Yaskawa INFORM job: BATMAN_4SPOINY.JBI

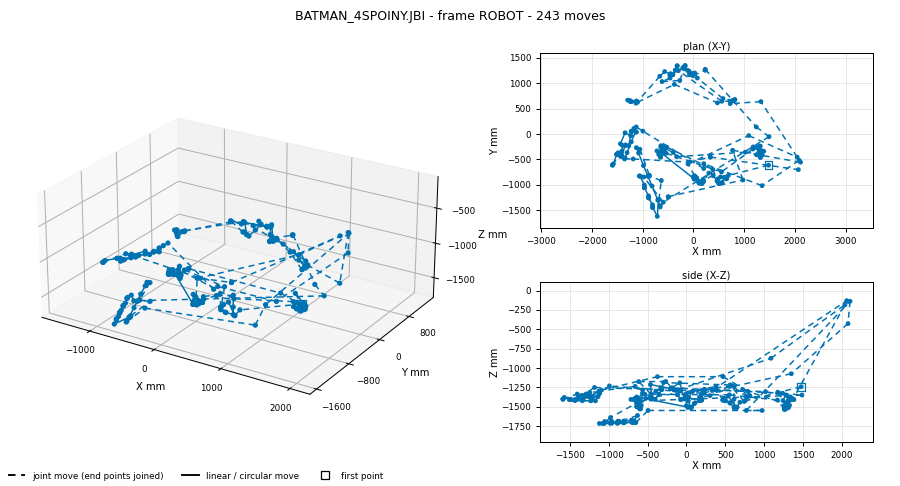
[picture p0: tool path of BATMAN_4SPOINY.JBI in frame ROBOT, 243 of 243 moves have a stored position in this frame; points joined in program order, loops and branches not executed]
/JOB
//NAME BATMAN_4SPOINY
///FOLDERNAME KRIS-SCIANA
//POS
///NPOS 293,293,243,19,0,0
///TOOL 0
///POSTYPE ROBOT
///RECTAN
///RCONF 0,0,0,0,0,0,0,0,0,0,0,0,0,0,0,0,0,0,0,0,0,0,0,0
C00000=1479.209,-614.254,-1239.827,11.6326,33.9671,-178.8219
C00001=689.483,-815.605,-1440.476,-6.5164,31.4559,38.6760
C00002=651.465,-878.509,-1502.529,-6.5193,31.4567,38.6726
C00003=649.681,-879.962,-1505.034,-6.5204,31.4570,38.6688
C00004=649.679,-879.971,-1512.967,-6.5216,31.4579,38.6721
C00005=649.681,-879.962,-1505.034,-6.5204,31.4570,38.6688
C00006=638.496,-885.487,-1507.904,-6.5213,31.4572,38.6690
C00007=649.681,-879.962,-1505.034,-6.5204,31.4570,38.6688
C00008=536.093,-844.110,-1358.224,-6.5194,31.4565,38.6698
C00009=485.208,-882.506,-1390.226,-6.5180,31.4566,38.6722
C00010=469.831,-925.588,-1412.310,-6.5196,31.4595,38.6720
C00011=469.838,-925.615,-1422.209,-6.5208,31.4607,38.6737
C00012=469.831,-925.588,-1412.310,-6.5196,31.4595,38.6720
C00013=460.916,-939.180,-1415.903,-6.5217,31.4610,38.6723
C00014=469.831,-925.588,-1412.310,-6.5196,31.4595,38.6720
C00015=390.944,-821.412,-1288.258,-6.5186,31.4593,38.6713
C00016=190.918,-901.981,-1343.686,6.6116,30.8402,128.8224
C00017=190.919,-901.974,-1384.308,6.6118,30.8401,128.8238
C00018=195.878,-934.762,-1411.685,6.6092,30.8405,128.8212
C00019=195.887,-934.767,-1420.325,6.6101,30.8407,128.8263
C00020=195.878,-934.762,-1411.685,6.6092,30.8405,128.8212
C00021=202.495,-948.084,-1414.851,6.6099,30.8403,128.8223
C00022=195.878,-934.762,-1411.685,6.6092,30.8405,128.8212
C00023=-1.386,-846.899,-1381.133,6.6069,30.8405,134.1399
C00024=-1.384,-846.902,-1485.292,6.6071,30.8406,134.1408
C00025=18.120,-884.199,-1503.049,6.6086,30.8410,134.1399
C00026=18.115,-884.194,-1511.506,6.6087,30.8409,134.1387
C00027=18.120,-884.199,-1503.049,6.6086,30.8410,134.1399
C00028=26.172,-895.008,-1505.663,6.6092,30.8415,134.1385
C00029=18.120,-884.199,-1503.049,6.6086,30.8410,134.1399
C00030=-641.458,-364.123,-1372.142,-0.2839,36.0778,31.9819
C00031=-662.744,-397.701,-1394.268,-0.2832,36.0779,31.9810
C00032=-662.752,-397.694,-1404.858,-0.2824,36.0779,31.9809
C00033=-662.744,-397.701,-1394.268,-0.2832,36.0779,31.9810
C00034=-686.425,-397.683,-1394.265,-0.2810,36.0766,31.9839
C00035=-662.744,-397.701,-1394.268,-0.2832,36.0779,31.9810
C00036=-625.948,-397.698,-1394.261,-0.2841,36.0782,31.9781
C00037=-625.925,-343.094,-1439.073,9.9613,47.0818,38.8274
C00038=-644.908,-343.069,-1439.106,9.9622,47.0802,38.8274
C00039=-625.925,-343.094,-1439.073,9.9613,47.0818,38.8274
C00040=-625.922,-343.099,-1464.884,9.9612,47.0818,38.8282
C00041=-625.925,-343.094,-1439.073,9.9613,47.0818,38.8274
C00042=-566.979,-310.222,-1326.381,23.2450,43.4420,-7.8391
C00043=-584.457,-249.104,-1485.810,23.2479,43.4563,-7.8306
C00044=-624.439,-249.091,-1480.215,23.2486,43.4554,-7.8315
C00045=-642.398,-249.105,-1480.200,23.2465,43.4549,-7.8334
C00046=-624.439,-249.091,-1480.215,23.2486,43.4554,-7.8315
C00047=-624.484,-249.097,-1506.745,23.2491,43.4587,-7.8307
C00048=-624.439,-249.091,-1480.215,23.2486,43.4554,-7.8315
C00049=-395.220,-362.676,-1299.812,-0.2837,36.0781,31.9812
C00050=-328.978,-445.538,-1251.827,-0.2820,36.0777,31.9846
C00051=1019.066,-358.271,-1303.588,-0.7093,36.3388,173.5111
C00052=1312.502,-388.638,-1368.088,-0.7090,36.3391,143.8761
C00053=1330.261,-409.263,-1395.611,-0.7097,36.3382,143.8752
C00054=1330.266,-409.258,-1408.665,-0.7105,36.3381,143.8742
C00055=1330.261,-409.263,-1395.611,-0.7097,36.3382,143.8752
C00056=1359.166,-409.282,-1395.624,-0.7081,36.3381,143.8755
C00057=1330.261,-409.263,-1395.611,-0.7097,36.3382,143.8752
C00058=1281.441,-409.290,-1348.405,-0.7080,36.3381,143.8761
C00059=1243.859,-409.326,-1418.007,-23.4626,32.8547,152.6563
C00060=1295.871,-355.597,-1446.808,-23.4629,32.8551,152.6521
C00061=1312.474,-355.618,-1446.814,-23.4633,32.8531,152.6491
C00062=1295.871,-355.597,-1446.808,-23.4629,32.8551,152.6521
C00063=1295.862,-355.607,-1467.339,-23.4610,32.8553,152.6551
C00064=1295.871,-355.597,-1446.808,-23.4629,32.8551,152.6521
C00065=1259.038,-270.785,-1482.658,-23.4624,32.8547,152.6509
C00066=1298.870,-254.314,-1488.573,-23.4632,32.8535,152.6493
C00067=1313.032,-254.323,-1488.569,-23.4626,32.8539,152.6494
C00068=1298.870,-254.314,-1488.573,-23.4632,32.8535,152.6493
C00069=1298.863,-254.294,-1509.572,-23.4652,32.8516,152.6464
C00070=1298.870,-254.314,-1488.573,-23.4632,32.8535,152.6493
C00071=1177.741,-254.308,-1309.531,-23.4643,32.8524,152.6474
C00072=1346.256,-330.236,-1377.208,-0.7085,36.3387,143.8760
C00073=1385.768,-339.505,-1405.683,-0.7074,36.3385,143.8819
C00074=1351.454,-409.571,-1404.855,-0.7093,36.3378,143.8750
C00075=1346.414,-413.349,-1407.345,-0.7117,36.3413,143.8740
C00076=1321.565,-460.935,-1406.687,-0.7131,36.3377,143.8716
C00077=1316.585,-457.113,-1411.355,-0.7151,36.3388,143.8640
C00078=1314.211,-431.828,-1419.878,-0.7170,36.3383,163.2059
C00079=1313.610,-343.846,-1457.563,-0.7163,36.3370,163.2057
C00080=1317.017,-236.585,-1505.551,-0.7181,36.3387,-169.8397
C00081=1305.403,-242.340,-1513.186,-0.7146,36.3426,-169.8375
C00082=1273.878,-260.855,-1530.310,-0.7179,36.3431,-169.8388
C00083=1267.455,-262.935,-1531.246,1.6686,33.5129,174.0872
C00084=1260.684,-274.038,-1530.726,2.4144,32.4266,168.8906
C00085=1172.939,-295.478,-1411.838,2.4149,32.4260,168.8924
C00086=553.926,-745.251,-1344.470,9.9580,22.3671,144.0884
C00087=-536.407,-379.228,-1337.930,-3.7346,30.6001,32.3556
C00088=-716.129,-331.806,-1403.803,-3.7368,30.5972,32.3471
C00089=-679.419,-400.533,-1403.776,-3.7326,30.5994,32.3503
C00090=-676.674,-401.500,-1405.574,-3.7338,30.5989,32.3549
C00091=-649.821,-454.382,-1404.684,-3.7317,30.5978,32.3601
C00092=-643.025,-452.350,-1408.275,-3.7303,30.5970,32.3639
C00093=-643.865,-446.825,-1410.310,-3.7312,30.5967,32.3587
C00094=-642.234,-424.038,-1414.216,6.8178,41.7169,38.5692
C00095=-644.123,-348.214,-1449.032,6.8176,41.7181,38.5693
C00096=-642.205,-255.965,-1492.156,6.7707,41.4319,23.5743
C00097=-637.301,-230.816,-1500.834,6.8206,41.7178,-9.7992
C00098=-602.821,-254.340,-1524.215,12.2915,40.7278,-6.2428
C00099=-595.514,-258.514,-1525.507,6.8184,41.7182,-9.7990
C00100=-591.339,-265.747,-1526.005,6.8213,41.7182,22.2664
C00101=-524.640,-257.672,-1391.051,6.8232,41.7195,-9.7941
C00102=380.759,-694.733,-1238.103,3.2707,31.6263,64.5290
C00103=500.376,-972.906,-1419.509,2.7673,30.8880,70.6771
C00104=502.727,-974.471,-1420.148,2.7642,30.8895,70.6782
C00105=558.221,-962.583,-1445.651,29.9139,35.7052,85.7904
C00106=565.911,-953.297,-1452.392,19.5066,42.2165,79.2495
C00107=613.155,-854.018,-1511.422,19.5140,42.2128,79.2557
C00108=613.159,-854.025,-1402.872,19.5132,42.2134,79.2549
C00109=613.167,-854.032,-1236.959,-5.3690,36.3099,63.2167
C00110=303.930,-769.190,-1354.154,12.5353,29.0330,117.3688
C00111=168.124,-974.808,-1376.941,12.5336,29.0302,117.3780
C00112=168.116,-974.806,-1418.609,12.5340,29.0299,117.3778
C00113=164.039,-975.283,-1418.603,12.5353,29.0308,117.3759
C00114=112.244,-968.180,-1447.281,-20.8953,38.2909,102.6892
C00115=98.759,-941.725,-1460.359,-8.8488,43.5839,114.0652
C00116=66.281,-869.518,-1502.684,-8.8494,43.5864,113.0954
C00117=58.364,-855.410,-1511.913,-8.8467,43.5844,111.1393
C00118=24.347,-822.026,-1422.241,-8.8464,43.5856,106.1673
C00119=-104.195,-589.697,-1279.272,-8.7711,29.7586,106.6768
C00120=1089.919,-31.439,-873.125,-36.7541,69.9873,137.0084
///RCONF 0,0,0,0,1,0,0,0,0,0,0,0,0,0,0,0,0,0,0,0,0,0,0,0
C00121=2042.728,-454.958,-183.433,1.6788,-19.8065,-6.7510
C00122=1329.047,637.602,-1479.857,8.0540,25.5528,30.8439
///RCONF 0,0,0,0,0,0,0,0,0,0,0,0,0,0,0,0,0,0,0,0,0,0,0,0
C00123=724.107,597.545,-1276.344,-3.2635,41.6684,-140.4024
C00124=785.383,659.459,-1372.820,-3.2632,41.6678,-140.4000
C00125=792.753,652.576,-1383.361,-3.2644,41.6697,-140.4060
C00126=785.383,659.459,-1372.820,-3.2632,41.6678,-140.4000
C00127=780.124,673.327,-1385.992,-3.2593,41.6675,-140.3923
C00128=785.383,659.459,-1372.820,-3.2632,41.6678,-140.4000
C00129=583.065,697.790,-1226.639,-3.1675,40.5415,-139.9875
C00130=78.541,1101.355,-1300.787,10.2599,31.0601,-45.0596
C00131=26.821,1201.359,-1372.636,10.2610,31.0614,-45.0581
C00132=-26.114,1184.722,-1395.825,10.2614,31.0609,-45.0571
C00133=-26.119,1184.747,-1409.910,10.2622,31.0622,-45.0567
C00134=-26.114,1184.722,-1395.825,10.2614,31.0609,-45.0571
C00135=-38.557,1201.364,-1401.881,10.2611,31.0613,-45.0602
C00136=-26.114,1184.722,-1395.825,10.2614,31.0609,-45.0571
C00137=-85.944,1239.452,-1189.279,10.2632,31.0602,-45.0547
C00138=-202.376,1302.359,-1263.326,10.2654,31.0601,-39.0783
C00139=-202.377,1302.375,-1273.759,10.2665,31.0600,-39.0755
C00140=-202.376,1302.359,-1263.326,10.2654,31.0601,-39.0783
C00141=-213.401,1315.412,-1266.159,10.2653,31.0594,-39.0754
C00142=-202.376,1302.359,-1263.326,10.2654,31.0601,-39.0783
C00143=-463.805,1156.888,-1211.984,5.4408,32.3182,-121.2144
C00144=-448.455,1180.872,-1396.312,5.4420,32.3182,-121.2130
C00145=-448.461,1180.875,-1405.887,5.4414,32.3181,-121.2136
C00146=-448.455,1180.872,-1396.312,5.4420,32.3182,-121.2130
C00147=-438.739,1194.365,-1399.533,5.4424,32.3182,-121.2152
C00148=-448.455,1180.872,-1396.312,5.4420,32.3182,-121.2130
C00149=-564.871,1229.171,-1282.403,5.4479,32.3214,-121.2108
C00150=-661.200,1136.351,-1235.695,5.4453,32.3209,-21.5885
C00151=-1128.608,606.997,-1296.811,5.4402,32.3220,-21.6018
C00152=-1245.560,650.345,-1363.191,5.4391,32.3216,-21.6043
C00153=-1253.840,659.612,-1369.532,5.4396,32.3086,-21.6048
C00154=-1245.560,650.345,-1363.191,5.4391,32.3216,-21.6043
C00155=-1255.518,641.298,-1375.299,5.4388,32.3217,-21.6053
C00156=-1245.560,650.345,-1363.191,5.4391,32.3216,-21.6043
C00157=-1122.499,650.360,-1312.804,5.4384,32.3212,-21.6061
C00158=-1246.019,650.333,-1312.805,-5.9814,50.4641,-44.8970
C00159=-1292.161,665.897,-1333.796,-5.9811,50.4635,-44.8938
C00160=-1228.051,636.266,-1400.155,-5.9792,50.4685,-44.8889
C00161=-1221.405,638.487,-1404.669,9.2040,37.0997,-34.2699
C00162=-1097.819,626.024,-1284.700,9.2046,37.0985,-34.2704
C00163=-374.253,977.072,-1110.582,-16.3615,18.9747,-168.4330
C00164=472.792,614.034,-1110.590,-6.3310,51.0848,-162.4334
C00165=790.077,666.826,-1299.714,-6.3326,51.0845,-162.4374
C00166=816.173,675.910,-1358.543,-6.3341,51.0842,-155.2649
C00167=816.189,675.286,-1355.228,-6.3386,51.0862,-155.2697
C00168=757.591,647.487,-1417.938,-6.3356,51.0871,-155.2637
C00169=745.147,646.476,-1430.103,-12.0666,41.5969,-159.4258
C00170=561.133,644.284,-1217.351,-12.0669,41.5966,-159.4267
C00171=-294.154,1247.220,-1186.692,-14.7086,35.8481,-158.3060
C00172=-317.097,1344.373,-1273.789,-9.3533,38.0929,-150.1876
C00173=-320.077,1338.543,-1279.711,-14.2234,35.5992,-165.4072
C00174=-357.428,1258.774,-1337.018,-14.2216,35.5960,-169.2182
C00175=-402.732,1164.520,-1402.173,-14.2202,35.5988,-165.9276
C00176=-458.281,1100.105,-1332.877,-14.2202,35.5995,-157.9829
C00177=-615.113,1031.882,-1174.072,-14.2237,35.6047,-144.5023
C00178=-266.790,1052.428,-1172.785,14.1594,35.6599,-52.4229
C00179=-185.740,1283.953,-1252.491,14.1602,35.6569,-52.4203
C00180=-163.350,1347.913,-1274.487,14.1614,35.6572,-52.4200
C00181=-161.403,1342.862,-1281.279,7.3802,43.3671,-41.1599
C00182=-113.870,1250.739,-1345.243,7.3795,43.3689,-41.1646
C00183=-75.578,1173.045,-1403.534,7.3827,43.3703,-41.1594
C00184=-71.378,1165.451,-1408.302,7.3856,43.3696,-41.1548
C00185=-4.180,1146.259,-1333.254,7.3847,43.3705,-41.1580
C00186=233.273,1258.338,-1276.378,4.6470,38.1496,-47.5838
C00187=233.273,1258.338,-1276.378,4.6470,38.1496,-47.5838
C00188=233.248,1273.531,-1276.386,4.6460,38.1499,-47.5825
C00189=1238.436,139.129,-1323.509,-1.5927,36.9682,-135.2428
C00190=1488.778,-52.476,-1347.695,27.2487,24.5669,-70.7938
C00191=-591.325,-1341.846,-1422.510,-0.6043,40.8297,16.7434
C00192=-978.344,-845.186,-1637.203,-0.6000,40.8277,16.7477
C00193=-1060.694,-827.545,-1707.801,-4.7604,28.0908,14.3911
C00194=-1060.693,-827.533,-1713.449,-4.7601,28.0909,14.3890
C00195=-1060.691,-827.539,-1712.151,-4.7601,28.0907,14.3910
C00196=-1067.726,-833.068,-1712.128,-4.7632,28.0919,14.3896
C00197=-1050.906,-827.500,-1697.143,-4.7577,28.0886,14.3917
C00198=-964.064,-1003.361,-1685.365,-0.5978,40.8280,16.7499
C00199=-963.616,-1055.856,-1701.250,-2.6259,23.7945,15.2047
C00200=-963.610,-1055.847,-1711.298,-2.6253,23.7935,15.2032
C00201=-963.602,-1055.842,-1710.131,-2.6247,23.7926,15.2047
C00202=-974.707,-1061.726,-1710.162,-2.6241,23.7909,15.2047
C00203=-963.602,-1055.860,-1700.361,-2.6260,23.7925,15.2034
C00204=-883.106,-1217.890,-1684.422,-0.5980,40.8275,16.7460
C00205=-880.117,-1256.561,-1698.940,-3.9703,31.1300,14.7591
C00206=-880.109,-1256.581,-1707.789,-3.9721,31.1294,14.7576
C00207=-880.105,-1256.591,-1706.390,-3.9730,31.1289,14.7563
C00208=-892.375,-1261.346,-1706.415,-3.9724,31.1284,14.7573
C00209=-880.093,-1256.566,-1697.766,-3.9719,31.1281,14.7561
C00210=-804.394,-1392.262,-1680.447,-0.5972,40.8269,16.7457
C00211=-801.090,-1443.591,-1697.691,-4.9918,27.6969,14.2534
C00212=-801.080,-1443.579,-1704.408,-4.9907,27.6963,14.2562
C00213=-801.094,-1443.589,-1702.814,-4.9912,27.6970,14.2539
C00214=-815.625,-1446.575,-1702.816,-4.9917,27.6963,14.2514
C00215=-801.096,-1443.607,-1692.082,-4.9930,27.6969,14.2499
C00216=-709.611,-1620.676,-1670.338,-0.5978,40.8273,16.7476
C00217=-687.434,-1294.732,-1692.603,-4.7533,28.5194,14.3647
C00218=-687.441,-1294.771,-1702.532,-4.7556,28.5199,14.3627
C00219=-687.456,-1294.784,-1700.544,-4.7557,28.5213,14.3651
C00220=-702.205,-1299.730,-1700.541,-4.7557,28.5223,14.3634
C00221=-678.347,-1292.883,-1678.457,-4.7568,28.5223,14.3642
C00222=-630.511,-916.030,-1610.753,-0.6017,40.8266,16.7401
C00223=-868.430,-829.435,-1692.124,-0.6028,40.8258,16.7353
C00224=-891.174,-831.785,-1707.986,-0.5978,40.8255,10.3627
C00225=-982.274,-621.589,-1711.536,-0.6040,40.8306,10.3525
C00226=-1078.436,-374.545,-1713.996,-0.6019,40.8306,10.3570
C00227=-1121.690,-268.616,-1714.197,-0.5999,40.8276,10.3556
C00228=-1052.650,-299.020,-1688.341,-0.6009,40.8211,16.7408
C00229=-865.284,-812.787,-1688.334,-0.6039,40.8202,42.9608
C00230=-893.481,-830.026,-1708.632,-0.5990,40.8174,42.9669
C00231=-813.172,-1023.978,-1705.511,-0.6003,40.8150,42.9585
C00232=-701.004,-1299.810,-1701.103,-0.6012,40.8175,42.9606
C00233=-658.788,-1411.167,-1701.911,-0.6004,40.8176,42.9675
C00234=-651.853,-1436.186,-1701.975,-0.5985,40.8188,42.9654
C00235=-495.179,-1232.483,-1546.245,-0.5800,40.8231,42.9777
C00236=975.318,-905.329,-1546.300,2.7447,40.6858,121.3068
C00237=771.357,-320.253,-1546.238,-0.5794,40.8236,124.0583
///RCONF 0,0,0,0,1,0,0,0,0,0,0,0,0,0,0,0,0,0,0,0,0,0,0,0
C00238=2108.910,-555.323,-138.194,2.1712,-19.6918,-3.5371
///RCONF 0,0,0,0,0,0,0,0,0,0,0,0,0,0,0,0,0,0,0,0,0,0,0,0
C00239=2082.559,-517.688,-426.187,17.7899,-11.9984,-30.1124
C00240=1351.715,-1016.627,-1072.730,14.7650,1.4143,-53.7135
C00241=205.703,-583.482,-1322.085,9.2825,24.4184,-95.9833
C00242=203.961,-679.195,-1324.426,-9.5613,21.9567,95.9050
C00243=-993.168,56.729,-1229.540,-0.2104,49.9239,-21.9207
C00244=-1124.976,139.813,-1330.335,5.3125,39.0598,-25.3648
C00245=-1217.958,48.598,-1401.440,5.3913,38.9364,-25.3168
C00246=-1222.465,48.743,-1409.263,5.3874,38.9378,-25.3223
C00247=-1222.459,48.730,-1420.612,5.3858,38.9371,-25.3242
C00248=-1222.465,48.743,-1409.263,5.3874,38.9378,-25.3223
C00249=-1239.080,48.748,-1409.236,5.3856,38.9399,-25.3266
C00250=-1222.465,48.743,-1409.263,5.3874,38.9378,-25.3223
C00251=-1271.414,-233.653,-1365.903,5.3880,38.9368,-25.3214
C00252=-1335.102,-218.968,-1407.739,5.3747,38.9270,-25.3244
C00253=-1335.110,-218.964,-1419.095,5.3738,38.9278,-25.3274
C00254=-1335.102,-218.968,-1407.739,5.3747,38.9270,-25.3244
C00255=-1351.938,-218.955,-1407.734,5.3749,38.9273,-25.3233
C00256=-1335.102,-218.968,-1407.739,5.3747,38.9270,-25.3244
C00257=-1410.796,-411.626,-1397.644,5.3751,38.9281,-25.3225
C00258=-1428.227,-437.232,-1406.270,5.3763,38.9287,-25.3214
C00259=-1428.230,-437.231,-1419.122,5.3758,38.9290,-25.3227
C00260=-1428.227,-437.232,-1406.270,5.3763,38.9287,-25.3214
C00261=-1445.183,-437.215,-1406.274,5.3770,38.9284,-25.3233
C00262=-1428.227,-437.232,-1406.270,5.3763,38.9287,-25.3214
C00263=-1478.764,-369.056,-1406.265,5.3746,38.9285,-25.3278
C00264=-1508.274,-399.507,-1403.549,5.3752,38.9282,-25.3298
C00265=-1508.284,-399.505,-1415.860,5.3764,38.9286,-25.3265
C00266=-1508.274,-399.507,-1403.549,5.3752,38.9282,-25.3298
C00267=-1525.499,-399.503,-1403.534,5.3741,38.9288,-25.3312
C00268=-1508.274,-399.507,-1403.549,5.3752,38.9282,-25.3298
C00269=-1573.700,-586.702,-1378.129,5.3749,38.9274,-25.3303
C00270=-1591.625,-610.872,-1399.727,5.3751,38.9284,-25.3300
C00271=-1591.607,-610.857,-1410.848,5.3774,38.9278,-25.3276
C00272=-1591.625,-610.872,-1399.727,5.3751,38.9284,-25.3300
C00273=-1607.585,-610.886,-1399.726,5.3748,38.9284,-25.3293
C00274=-1591.625,-610.872,-1399.727,5.3751,38.9284,-25.3300
C00275=-1407.614,-340.295,-1334.283,5.3763,38.9277,-25.3283
C00276=-1393.545,-225.421,-1380.034,5.3755,38.9268,-25.3271
C00277=-1436.319,-192.923,-1419.519,-0.6441,37.4048,-43.4681
C00278=-1343.970,24.204,-1419.685,-0.6458,37.4045,-43.4729
C00279=-1233.172,-33.364,-1421.676,-0.6450,37.4042,-43.4706
C00280=-1172.683,108.529,-1421.468,-0.6415,37.4057,-43.4715
C00281=-1123.867,39.567,-1327.748,-0.6454,37.4059,-43.4725
C00282=-1123.867,39.567,-1327.748,-0.6454,37.4059,-43.4725
C00283=-1139.614,46.545,-1367.957,-0.6485,37.4091,-15.9314
C00284=-1221.149,-154.590,-1364.989,-0.6505,37.4071,-15.9367
C00285=-1304.293,-367.690,-1359.056,-0.6521,37.4085,-15.9430
C00286=-1343.286,-469.596,-1355.805,-0.6535,37.4062,-15.9492
C00287=-1354.672,-491.189,-1354.002,-0.6534,37.4048,-15.9508
C00288=-1184.082,-491.180,-1249.860,-0.6521,37.4040,-15.9519
C00289=-78.969,-554.378,-1286.716,1.4249,23.3229,2.1506
C00290=333.912,-453.248,-1285.762,1.2790,23.3311,46.5433
C00291=333.896,-453.245,-1285.777,1.2802,23.3310,46.5456
C00292=2065.993,-701.065,-130.284,1.6748,-19.7957,-6.8086
BC00000=506.026,2197.799,889.024
BC00001=1028.973,2071.524,879.905
BC00002=1028.973,2071.524,879.905
BC00003=1028.973,2071.524,879.905
BC00004=1028.973,2071.524,879.905
BC00005=1028.973,2071.524,879.905
BC00006=1028.973,2071.524,879.905
BC00007=1028.973,2071.524,879.905
BC00008=1028.973,2071.524,879.905
BC00009=1028.973,2071.524,879.905
BC00010=1028.973,2071.524,879.905
BC00011=1028.973,2071.524,879.905
BC00012=1028.973,2071.524,879.905
BC00013=1028.973,2071.524,879.905
BC00014=1028.973,2071.524,879.905
BC00015=1028.973,2071.524,879.905
BC00016=1028.973,2071.524,879.905
BC00017=1028.973,2071.524,879.905
BC00018=1028.973,2071.524,879.905
BC00019=1028.973,2071.524,879.905
BC00020=1028.973,2071.524,879.905
BC00021=1028.973,2071.524,879.905
BC00022=1028.973,2071.524,879.905
BC00023=1028.973,2071.524,879.905
BC00024=1028.973,2071.524,879.905
BC00025=1028.973,2071.524,879.905
BC00026=1028.973,2071.524,879.905
BC00027=1028.973,2071.524,879.905
BC00028=1028.973,2071.524,879.905
BC00029=1028.973,2071.524,879.905
BC00030=1028.973,2071.524,879.905
BC00031=1028.973,2071.524,879.905
BC00032=1028.973,2071.524,879.905
BC00033=1028.973,2071.524,879.905
BC00034=1028.973,2071.524,879.905
BC00035=1028.973,2071.524,879.905
BC00036=1028.973,2071.524,879.905
BC00037=1028.973,2071.524,879.905
BC00038=1028.973,2071.524,879.905
BC00039=1028.973,2071.524,879.905
BC00040=1028.973,2071.524,879.905
BC00041=1028.973,2071.524,879.905
BC00042=1028.966,2071.524,879.901
BC00043=1028.966,2071.531,879.892
BC00044=1028.966,2071.531,879.892
BC00045=1028.966,2071.531,879.892
BC00046=1028.966,2071.531,879.892
BC00047=1028.966,2071.531,879.892
BC00048=1028.966,2071.531,879.892
BC00049=1028.973,2071.524,879.905
BC00050=1028.973,2071.524,879.905
BC00051=1028.973,2071.524,879.905
BC00052=1028.973,2071.524,879.905
BC00053=1028.973,2071.524,879.905
BC00054=1028.973,2071.524,879.905
BC00055=1028.973,2071.524,879.905
BC00056=1028.973,2071.524,879.905
BC00057=1028.973,2071.524,879.905
BC00058=1028.973,2071.524,879.905
BC00059=1028.973,2071.524,879.905
BC00060=1028.973,2071.524,879.905
BC00061=1028.973,2071.524,879.905
BC00062=1028.973,2071.524,879.905
BC00063=1028.973,2071.524,879.905
BC00064=1028.973,2071.524,879.905
BC00065=1028.973,2071.524,879.905
BC00066=1028.973,2071.524,879.905
BC00067=1028.973,2071.524,879.905
BC00068=1028.973,2071.524,879.905
BC00069=1028.973,2071.524,879.905
BC00070=1028.973,2071.524,879.905
BC00071=1028.973,2071.524,879.905
BC00072=1028.973,2071.524,879.905
BC00073=1028.973,2071.524,879.905
BC00074=1028.973,2071.524,879.905
BC00075=1028.973,2071.524,879.905
BC00076=1028.973,2071.524,879.905
BC00077=1028.973,2071.524,879.905
BC00078=1028.973,2071.524,879.905
BC00079=1028.973,2071.524,879.905
BC00080=1028.973,2071.524,879.905
BC00081=1028.973,2071.524,879.905
BC00082=1028.973,2071.524,879.905
BC00083=1028.979,2071.524,879.911
BC00084=1028.979,2071.524,879.911
BC00085=1028.979,2071.524,879.911
BC00086=1028.979,2071.531,1132.335
BC00087=1028.979,2071.531,879.905
BC00088=1028.979,2071.531,879.905
BC00089=1028.979,2071.531,879.905
BC00090=1028.979,2071.531,879.905
BC00091=1028.979,2071.531,879.905
BC00092=1028.979,2071.531,879.905
BC00093=1028.979,2071.531,879.905
BC00094=1028.979,2071.531,879.905
BC00095=1028.979,2071.531,879.905
BC00096=1028.979,2071.531,879.905
BC00097=1028.979,2071.531,879.905
BC00098=1028.979,2071.531,879.905
BC00099=1028.979,2071.531,879.905
BC00100=1028.979,2071.531,879.905
BC00101=1028.979,2071.531,879.905
BC00102=1028.979,2071.531,879.905
BC00103=1028.979,2071.531,879.905
BC00104=1028.979,2071.531,879.905
BC00105=1028.979,2071.531,879.905
BC00106=1028.979,2071.531,879.905
BC00107=1028.979,2071.531,879.905
BC00108=1028.979,2071.531,879.905
BC00109=1028.979,2071.531,879.905
BC00110=1028.979,2071.531,879.905
BC00111=1028.979,2071.531,879.905
BC00112=1028.979,2071.531,879.905
BC00113=1028.979,2071.531,879.905
BC00114=1028.979,2071.531,879.905
BC00115=1028.979,2071.531,879.905
BC00116=1028.979,2071.531,879.905
BC00117=1028.979,2071.531,879.905
BC00118=1028.979,2071.531,879.905
BC00119=1028.979,2071.531,1313.400
BC00120=705.175,35.017,1952.866
BC00121=786.422,38.780,1999.645
BC00122=786.422,38.780,1999.645
BC00123=1602.623,32.856,1148.414
BC00124=1602.623,32.856,1148.414
BC00125=1602.623,32.856,1148.414
BC00126=1602.623,32.856,1148.414
BC00127=1602.623,32.856,1148.414
BC00128=1602.623,32.856,1148.414
BC00129=1602.623,32.856,1148.414
BC00130=1602.623,32.856,1148.414
BC00131=1602.623,32.856,1148.414
BC00132=1602.623,32.856,1148.414
BC00133=1602.623,32.856,1148.414
BC00134=1602.623,32.856,1148.414
BC00135=1602.623,32.856,1148.414
BC00136=1602.623,32.856,1148.414
BC00137=1602.623,32.856,1148.414
BC00138=1602.623,32.856,1148.414
BC00139=1602.623,32.856,1148.414
BC00140=1602.623,32.856,1148.414
BC00141=1602.623,32.856,1148.414
BC00142=1602.623,32.856,1148.414
BC00143=1602.623,32.856,1148.414
BC00144=1602.623,32.856,1148.414
BC00145=1602.623,32.856,1148.414
BC00146=1602.623,32.856,1148.414
BC00147=1602.623,32.856,1148.414
BC00148=1602.623,32.856,1148.414
BC00149=1602.623,32.856,1148.414
BC00150=1602.623,32.856,1148.414
BC00151=1602.623,32.856,1148.414
BC00152=1602.623,32.856,1148.414
BC00153=1602.617,32.863,1148.408
BC00154=1602.623,32.856,1148.414
BC00155=1602.623,32.856,1148.414
BC00156=1602.623,32.856,1148.414
BC00157=1602.623,32.856,1148.414
BC00158=1602.623,32.856,1148.414
BC00159=1602.623,32.856,1148.414
BC00160=1602.623,32.856,1148.414
BC00161=1602.623,32.856,1148.414
BC00162=1602.623,32.856,1148.414
BC00163=1602.617,32.856,1148.408
BC00164=1602.617,32.856,1148.408
BC00165=1602.617,32.856,1148.408
BC00166=1602.617,32.856,1148.408
BC00167=1602.610,32.863,1148.395
BC00168=1602.610,32.863,1148.395
BC00169=1602.610,32.863,1148.395
BC00170=1602.610,32.863,1148.395
BC00171=1602.610,32.863,1148.395
BC00172=1602.610,32.863,1148.391
BC00173=1602.610,32.863,1148.391
BC00174=1602.610,32.863,1148.391
BC00175=1602.610,32.863,1148.391
BC00176=1602.610,32.863,1148.391
BC00177=1602.610,32.863,1148.391
BC00178=1602.610,32.863,1148.391
BC00179=1602.617,32.863,1148.387
BC00180=1602.617,32.863,1148.387
BC00181=1602.617,32.863,1148.387
BC00182=1602.617,32.863,1148.387
BC00183=1602.617,32.863,1148.387
BC00184=1602.617,32.863,1148.387
BC00185=1602.617,32.863,1148.387
BC00186=1602.617,32.863,1960.335
BC00187=2287.550,32.863,1960.335
BC00188=2172.832,3214.278,1960.335
BC00189=752.940,3214.278,1960.335
BC00190=766.746,3215.828,1976.542
BC00191=1984.483,3218.041,658.883
BC00192=1984.483,2448.792,658.883
BC00193=1984.483,2448.792,658.883
BC00194=1984.483,2448.792,658.883
BC00195=1984.483,2448.792,658.883
BC00196=1984.483,2448.792,658.883
BC00197=1984.483,2448.792,658.883
BC00198=1984.483,2448.792,658.883
BC00199=1984.483,2448.792,658.883
BC00200=1984.483,2448.792,658.883
BC00201=1984.483,2448.792,658.883
BC00202=1984.483,2448.792,658.883
BC00203=1984.483,2448.792,658.883
BC00204=1984.483,2448.792,658.883
BC00205=1984.483,2448.792,658.883
BC00206=1984.483,2448.792,658.883
BC00207=1984.483,2448.792,658.883
BC00208=1984.483,2448.792,658.883
BC00209=1984.483,2448.792,658.883
BC00210=1984.483,2448.792,658.883
BC00211=1984.483,2448.792,658.883
BC00212=1984.483,2448.792,658.883
BC00213=1984.483,2448.792,658.883
BC00214=1984.483,2448.792,658.883
BC00215=1984.483,2448.792,658.883
BC00216=1984.483,2448.792,658.883
BC00217=1984.483,2020.544,658.883
BC00218=1984.483,2020.544,658.883
BC00219=1984.483,2020.544,658.883
BC00220=1984.483,2020.544,658.883
BC00221=1984.483,2020.544,658.883
BC00222=1984.483,2020.544,658.883
BC00223=1984.483,2020.544,658.883
BC00224=1984.470,2020.544,658.879
BC00225=1984.470,2020.544,658.879
BC00226=1984.470,2020.544,658.879
BC00227=1984.470,2020.544,658.879
BC00228=1984.470,2020.544,658.879
BC00229=1984.470,2020.544,658.879
BC00230=1984.470,2020.544,658.879
BC00231=1984.470,2020.544,658.879
BC00232=1984.470,2020.544,658.879
BC00233=1984.470,2020.544,658.879
BC00234=1984.470,2020.544,658.879
BC00235=1984.470,2020.538,658.877
BC00236=1391.860,3285.602,1013.728
BC00237=874.011,3770.839,1827.894
BC00238=779.962,3777.824,1999.134
BC00239=536.351,3774.159,1979.823
BC00240=1536.650,3350.624,1880.104
BC00241=2471.115,2623.215,1708.837
BC00242=2471.115,644.771,1708.837
BC00243=2471.115,644.771,371.374
BC00244=2499.895,888.831,371.374
BC00245=2499.895,888.831,371.366
BC00246=2499.895,888.831,371.366
BC00247=2499.895,888.831,371.366
BC00248=2499.895,888.831,371.366
BC00249=2499.895,888.831,371.366
BC00250=2499.895,888.831,371.366
BC00251=2499.895,888.831,371.366
BC00252=2499.895,888.825,371.363
BC00253=2499.895,888.825,371.363
BC00254=2499.895,888.825,371.363
BC00255=2499.895,888.825,371.363
BC00256=2499.895,888.825,371.363
BC00257=2499.895,888.825,371.363
BC00258=2499.895,888.825,371.363
BC00259=2499.895,888.825,371.363
BC00260=2499.895,888.825,371.363
BC00261=2499.895,888.825,371.363
BC00262=2499.895,888.825,371.363
BC00263=2499.895,648.814,371.363
BC00264=2499.895,648.814,371.363
BC00265=2499.895,648.814,371.363
BC00266=2499.895,648.814,371.363
BC00267=2499.895,648.814,371.363
BC00268=2499.895,648.814,371.363
BC00269=2499.895,648.814,371.363
BC00270=2499.895,648.814,371.363
BC00271=2499.895,648.814,371.363
BC00272=2499.895,648.814,371.363
BC00273=2499.895,648.814,371.363
BC00274=2499.895,648.814,371.363
BC00275=2499.895,648.814,371.363
BC00276=2499.895,648.814,371.363
BC00277=2499.895,648.814,371.363
BC00278=2499.895,648.814,371.363
BC00279=2499.895,972.335,371.363
BC00280=2499.895,972.335,371.363
BC00281=2499.895,972.335,371.363
BC00282=2204.921,409.519,319.294
BC00283=2204.921,409.519,319.294
BC00284=2204.921,409.519,319.294
BC00285=2204.921,409.519,319.294
BC00286=2204.921,409.519,319.294
BC00287=2204.921,409.519,319.294
BC00288=2204.921,409.519,319.294
BC00289=2493.165,409.519,1451.480
BC00290=2493.165,3204.728,1451.480
BC00291=2493.165,3204.728,1451.476
BC00292=430.297,4179.635,1999.619
///POSTYPE PULSE
///PULSE
EC00000=-811452,-554689
EC00001=-811450,-554689
EC00002=-811450,-554689
EC00003=-811450,-554689
EC00004=-811450,-554689
EC00005=-811450,-554689
EC00006=-811450,-554689
EC00007=-811450,-554689
EC00008=-811450,-554689
EC00009=-811450,-554689
EC00010=-811450,-554689
EC00011=-811450,-554689
EC00012=-811450,-554689
EC00013=-811450,-554689
EC00014=-811450,-554689
EC00015=-811450,-554689
EC00016=-811450,-554689
EC00017=-811450,-554689
EC00018=-811450,-554689
EC00019=-811450,-554689
EC00020=-811450,-554689
EC00021=-811450,-554689
EC00022=-811450,-554689
EC00023=-811450,-554689
EC00024=-811450,-554689
EC00025=-811450,-554689
EC00026=-811450,-554689
EC00027=-811450,-554689
EC00028=-811450,-554689
EC00029=-811450,-554689
EC00030=-811447,-554690
EC00031=-811443,-554690
EC00032=-811443,-554690
EC00033=-811443,-554690
EC00034=-811443,-554690
EC00035=-811450,-554689
EC00036=-811450,-554689
EC00037=-811450,-554689
EC00038=-811450,-554689
EC00039=-811450,-554689
EC00040=-811450,-554689
EC00041=-811450,-554689
EC00042=-811450,-554689
EC00043=-811450,-554689
EC00044=-811450,-554689
EC00045=-811450,-554689
EC00046=-811450,-554689
EC00047=-811450,-554689
EC00048=-811450,-554689
EC00049=-811450,-554689
EC00050=-811450,-554689
EC00051=-811450,-554689
EC00052=-811450,-554689
EC00053=-811450,-554689
EC00054=-811450,-554689
EC00055=-811450,-554689
EC00056=-811450,-554689
EC00057=-811450,-554689
EC00058=-811450,-554689
EC00059=-811450,-554689
EC00060=-811450,-554689
EC00061=-811450,-554689
EC00062=-811450,-554689
EC00063=-811452,-554689
EC00064=-811452,-554689
EC00065=-811452,-554689
EC00066=-811451,-554689
EC00067=-811451,-554689
EC00068=-811451,-554689
EC00069=-811451,-554689
EC00070=-811451,-554689
EC00071=-811451,-554689
EC00072=-811451,-554689
EC00073=-811451,-554689
EC00074=-811451,-554689
EC00075=-811451,-554689
EC00076=-811451,-554689
EC00077=-811451,-554689
EC00078=-811451,-554689
EC00079=-811451,-554689
EC00080=-811451,-554689
EC00081=-811451,-554689
EC00082=-811451,-554689
EC00083=-811451,-554689
EC00084=-811451,-554689
EC00085=-811451,-554689
EC00086=-811451,-554689
EC00087=-811451,-554689
EC00088=-811451,-554689
EC00089=-811451,-554689
EC00090=-811451,-554689
EC00091=-811451,-554689
EC00092=-811451,-554689
EC00093=-811451,-554689
EC00094=-811451,-554689
EC00095=-811451,-554689
EC00096=-811451,-554689
EC00097=-811451,-554689
EC00098=-811451,-554689
EC00099=-811451,-554689
EC00100=-363208,-550746
EC00101=-363208,-550746
EC00102=-363208,-550746
EC00103=-363208,-550746
EC00104=-363208,-550746
EC00105=-363208,-550746
EC00106=-363208,-550746
EC00107=-363208,-550746
EC00108=-363208,-550746
EC00109=-363208,-550746
EC00110=-363208,-550746
EC00111=-363208,-550746
EC00112=-363208,-550746
EC00113=-363208,-550746
EC00114=-363208,-550746
EC00115=-363208,-550746
EC00116=-363208,-550746
EC00117=-363208,-550746
EC00118=-363208,-550746
EC00119=-363208,-550746
EC00120=-363208,-550746
EC00121=-363208,-550746
EC00122=-363208,-550746
EC00123=-363208,-550746
EC00124=-363208,-550746
EC00125=-363208,-550746
EC00126=-363208,-550746
EC00127=-363208,-550746
EC00128=-363208,-550746
EC00129=-363208,-550746
EC00130=-363208,-550746
EC00131=-363208,-550746
EC00132=-363208,-550746
EC00133=-363208,-550746
EC00134=-363208,-550746
EC00135=-363208,-550746
EC00136=-363208,-550746
EC00137=-363207,-550746
EC00138=-363207,-550746
EC00139=-363207,-550746
EC00140=-363207,-550746
EC00141=-363207,-550746
EC00142=-363206,-550746
EC00143=-363206,-550746
EC00144=-363206,-550746
EC00145=-363206,-550746
EC00146=-363206,-550746
EC00147=-363206,-550746
EC00148=-363206,-550746
EC00149=-363206,-550746
EC00150=-363206,-550746
EC00151=-363206,-550746
EC00152=-363206,-550746
EC00153=-363206,-550746
EC00154=-363206,-550746
EC00155=-363206,-550746
EC00156=-363206,-550746
EC00157=-363206,-550746
EC00158=0,0
EC00159=-802750,0
EC00160=-802750,0
EC00161=-802750,0
EC00162=-802750,0
EC00163=-802750,0
EC00164=-802750,0
EC00165=-802750,0
EC00166=-802750,0
EC00167=-802750,0
EC00168=-802750,0
EC00169=-802750,0
EC00170=-802750,0
EC00171=-802750,0
EC00172=-802750,0
EC00173=-802750,0
EC00174=-802750,0
EC00175=-802750,0
EC00176=-802750,0
EC00177=-802750,0
EC00178=-802750,0
EC00179=-802750,0
EC00180=-802750,0
EC00181=-802750,0
EC00182=-802750,0
EC00183=-802750,0
EC00184=-802749,0
EC00185=-802749,0
EC00186=-802749,0
EC00187=-802749,0
EC00188=-802749,0
EC00189=-802749,0
EC00190=-802749,0
EC00191=-802749,0
EC00192=-802749,0
EC00193=-802749,0
EC00194=-802749,0
EC00195=-802748,0
EC00196=-802748,0
EC00197=793507,0
EC00198=793506,-1
EC00199=793506,-1
EC00200=793506,-1
EC00201=793506,-1
EC00202=793506,-1
EC00203=793506,-1
EC00204=793506,-1
EC00205=793505,-1
EC00206=793505,-1
EC00207=793505,-1
EC00208=793505,-1
EC00209=793505,-1
EC00210=793504,-1
EC00211=793504,-1
EC00212=793504,-1
EC00213=793504,-1
EC00214=793504,-1
EC00215=793504,-1
EC00216=793504,-1
EC00217=793504,-1
EC00218=793504,-1
EC00219=793504,-1
EC00220=793504,-1
EC00221=793504,-1
EC00222=793504,-1
EC00223=793504,-1
EC00224=793504,-1
EC00225=793504,-1
EC00226=793504,-1
EC00227=793504,-1
EC00228=793504,-1
EC00229=793504,-1
EC00230=793504,-1
EC00231=793504,-1
EC00232=793504,-1
EC00233=793504,-1
EC00234=793504,-1
EC00235=793504,-1
EC00236=793504,-1
EC00237=793504,-1
EC00238=793504,-1
EC00239=793504,-1
EC00240=793504,-1
EC00241=793503,548424
EC00242=0,-1
///POSTYPE BASE
///RECTAN
///RCONF 0,0,0,0,1,0,0,0,0,0,0,0,0,0,0,0,0,0,0,0,0,0,0,0
P00006=2.006,1.622,-0.565,0.0000,0.0000,0.0000
P00021=0.073,2.058,-0.109,0.0000,0.0000,0.0000
P00022=2.006,1.622,-0.565,0.0000,0.0000,0.0000
///RCONF 0,0,0,0,0,0,0,0,0,0,0,0,0,0,0,0,0,0,0,0,0,0,0,0
P00023=-2.957,-4.083,2.762,0.0000,0.0000,0.0000
P00024=-1.466,-0.226,-0.419,0.0000,0.0000,0.0000
P00025=3.643,0.007,-2.585,0.0000,0.0000,0.0000
P00026=2.644,0.055,-2.583,0.0000,0.0000,0.0000
P00027=2.278,0.099,-4.210,0.0000,0.0000,0.0000
P00028=-1.778,-0.182,-2.050,0.0000,0.0000,0.0000
P00029=1.749,4.006,-0.261,0.0000,0.0000,0.0000
P00030=-0.014,-0.768,0.131,0.0000,0.0000,0.0000
///RCONF 0,0,0,0,1,0,0,0,0,0,0,0,0,0,0,0,0,0,0,0,0,0,0,0
P00034=-8.151,9.743,-4.393,0.0000,0.0000,0.0000
///RCONF 0,0,0,0,0,0,0,0,0,0,0,0,0,0,0,0,0,0,0,0,0,0,0,0
P00035=0.390,-0.027,1.040,0.0000,0.0000,0.0000
P00036=-2.434,0.084,0.197,0.0000,0.0000,0.0000
P00037=-1.075,5.090,-3.949,0.0000,0.0000,0.0000
P00040=2.716,-0.016,3.014,0.0000,0.0000,0.0000
P00041=-0.109,0.014,0.966,0.0000,0.0000,0.0000
P00042=-0.220,0.371,-0.613,0.0000,0.0000,0.0000
P00043=-0.179,-5.890,-3.227,0.0000,0.0000,0.0000
//INST
///DATE 2024/09/05 12:58
///ATTR SC,RW,RJ
////FRAME ROBOT
///GROUP1 RB1,BS1
///GROUP2 ST1
NOP
SFTOF
MOVJ C00000 BC00000 VJ=100.00  +MOVJ EC00000 VJ=100.00
'SZUKANIE
SFTOF
MOVJ C00001 BC00001 VJ=100.00  +MOVJ EC00001 VJ=30.00
MOVL C00002 BC00002 V=83.3  +MOVJ EC00002 VJ=15.00
MOVL C00003 BC00003 V=83.3  +MOVJ EC00003 VJ=15.00
REFP 3 RB1 C00004 BC00004
CALL JOB:SEARCH-R1
SET P026 P006
SFTON P026
MOVL C00005 BC00005 V=83.3  +MOVJ EC00004 VJ=15.00
REFP 3 RB1 C00006 BC00006
CALL JOB:SEARCH-R1
SET P026 P006
MOVL C00007 BC00007 V=83.3  +MOVJ EC00005 VJ=15.00
SFTOF
MOVL C00008 BC00008 V=83.3  +MOVJ EC00006 VJ=15.00
MOVL C00009 BC00009 V=83.3  +MOVJ EC00007 VJ=15.00
MOVL C00010 BC00010 V=83.3  +MOVJ EC00008 VJ=15.00
REFP 3 RB1 C00011 BC00011
CALL JOB:SEARCH-R1
SET P027 P006
SFTON P027
MOVL C00012 BC00012 V=83.3  +MOVJ EC00009 VJ=15.00
REFP 3 RB1 C00013 BC00013
CALL JOB:SEARCH-R1
SET P027 P006
MOVL C00014 BC00014 V=83.3  +MOVJ EC00010 VJ=15.00
SFTOF
MOVJ C00015 BC00015 VJ=100.00  +MOVJ EC00011 VJ=100.00
SFTOF
MOVJ C00016 BC00016 VJ=100.00  +MOVJ EC00012 VJ=100.00
MOVL C00017 BC00017 V=83.3  +MOVJ EC00013 VJ=15.00
MOVL C00018 BC00018 V=83.3  +MOVJ EC00014 VJ=15.00
REFP 3 RB1 C00019 BC00019
CALL JOB:SEARCH-R1
SET P029 P006
SFTON P029
MOVL C00020 BC00020 V=83.3  +MOVJ EC00015 VJ=15.00
REFP 3 RB1 C00021 BC00021
CALL JOB:SEARCH-R1
SET P029 P006
MOVL C00022 BC00022 V=83.3  +MOVJ EC00016 VJ=15.00
SFTOF
MOVL C00023 BC00023 V=83.3  +MOVJ EC00017 VJ=15.00
MOVL C00024 BC00024 V=83.3  +MOVJ EC00018 VJ=15.00
MOVL C00025 BC00025 V=83.3  +MOVJ EC00019 VJ=15.00
REFP 3 RB1 C00026 BC00026
CALL JOB:SEARCH-R1
SET P030 P006
SFTON P030
MOVL C00027 BC00027 V=83.3  +MOVJ EC00020 VJ=15.00
REFP 3 RB1 C00028 BC00028
CALL JOB:SEARCH-R1
SET P030 P006
MOVL C00029 BC00029 V=83.3  +MOVJ EC00021 VJ=15.00
SFTOF
MOVL C00030 BC00030 V=250.0  +MOVJ EC00022 VJ=15.00
MOVL C00031 BC00031 V=83.3  +MOVJ EC00023 VJ=15.00
REFP 3 RB1 C00032 BC00032
CALL JOB:SEARCH-R1
SET P036 P006
SFTON P036
MOVL C00033 BC00033 V=83.3  +MOVJ EC00024 VJ=15.00
REFP 3 RB1 C00034 BC00034
CALL JOB:SEARCH-R1
SET P036 P006
MOVL C00035 BC00035 V=83.3  +MOVJ EC00025 VJ=15.00
SFTOF
MOVL C00036 BC00036 V=11.0  +MOVJ EC00026 VJ=0.78
MOVL C00037 BC00037 V=83.3  +MOVJ EC00027 VJ=15.00
REFP 3 RB1 C00038 BC00038
CALL JOB:SEARCH-R1
SET P040 P006
SFTON P040
MOVL C00039 BC00039 V=83.3  +MOVJ EC00028 VJ=15.00
REFP 3 RB1 C00040 BC00040
CALL JOB:SEARCH-R1
SET P040 P006
MOVL C00041 BC00041 V=83.3  +MOVJ EC00029 VJ=15.00
SFTOF
MOVJ C00042 BC00042 VJ=100.00  +MOVJ EC00030 VJ=0.78
MOVJ C00043 BC00043 VJ=100.00  +MOVJ EC00031 VJ=100.00
MOVL C00044 BC00044 V=83.3  +MOVJ EC00032 VJ=15.00
REFP 3 RB1 C00045 BC00045
CALL JOB:SEARCH-R1
SET P041 P006
SFTON P041
MOVL C00046 BC00046 V=83.3  +MOVJ EC00033 VJ=15.00
REFP 3 RB1 C00047 BC00047
CALL JOB:SEARCH-R1
SET P041 P006
MOVL C00048 BC00048 V=83.3  +MOVJ EC00034 VJ=15.00
SFTOF
MOVL C00049 BC00049 V=250.0  +MOVJ EC00035 VJ=15.00
MOVJ C00050 BC00050 VJ=100.00  +MOVJ EC00036 VJ=15.00
MOVJ C00051 BC00051 VJ=100.00  +MOVJ EC00037 VJ=100.00
MOVJ C00052 BC00052 VJ=100.00  +MOVJ EC00038 VJ=100.00
MOVL C00053 BC00053 V=83.3  +MOVJ EC00039 VJ=15.00
REFP 3 RB1 C00054 BC00054
CALL JOB:SEARCH-R1
SET P037 P006
SFTON P037
MOVL C00055 BC00055 V=83.3  +MOVJ EC00040 VJ=15.00
REFP 3 RB1 C00056 BC00056
CALL JOB:SEARCH-R1
SET P037 P006
MOVL C00057 BC00057 V=83.3  +MOVJ EC00041 VJ=15.00
MOVJ C00058 BC00058 VJ=100.00  +MOVJ EC00042 VJ=100.00
MOVJ C00059 BC00059 VJ=100.00  +MOVJ EC00043 VJ=100.00
MOVL C00060 BC00060 V=83.3  +MOVJ EC00044 VJ=15.00
REFP 3 RB1 C00061 BC00061
CALL JOB:SEARCH-R1
SET P042 P006
SFTOF
SFTON P042
MOVL C00062 BC00062 V=83.3  +MOVJ EC00045 VJ=15.00
REFP 3 RB1 C00063 BC00063
CALL JOB:SEARCH-R1
SET P042 P006
MOVL C00064 BC00064 V=83.3  +MOVJ EC00046 VJ=15.00
SFTOF
MOVJ C00065 BC00065 VJ=100.00  +MOVJ EC00047 VJ=100.00
MOVL C00066 BC00066 V=83.3  +MOVJ EC00048 VJ=15.00
REFP 3 RB1 C00067 BC00067
CALL JOB:SEARCH-R1
SET P042 P006
SFTON P042
MOVL C00068 BC00068 V=83.3  +MOVJ EC00049 VJ=15.00
REFP 3 RB1 C00069 BC00069
CALL JOB:SEARCH-R1
SET P042 P006
MOVL C00070 BC00070 V=83.3  +MOVJ EC00050 VJ=15.00
SFTOF
MOVJ C00071 BC00071 VJ=100.00  +MOVJ EC00051 VJ=100.00
SFTOF
MOVL C00072 BC00072 V=166.7  +MOVJ EC00052 VJ=15.00
SFTON P037
MACRO1 MJ#(0) ARGF7
MOVL C00073 BC00073 V=83.3  +MOVJ EC00053 VJ=100.00
ARCON
MOVL C00074 BC00074 V=10.0  +MOVJ EC00054 VJ=100.00
MOVL C00075 BC00075 V=10.0  +MOVJ EC00055 VJ=100.00
MOVL C00076 BC00076 V=10.0  +MOVJ EC00056 VJ=100.00
MOVL C00077 BC00077 V=10.0  +MOVJ EC00057 VJ=100.00
MOVL C00078 BC00078 V=10.0  +MOVJ EC00058 VJ=100.00
SFTOF
SFTON P042
MOVL C00079 BC00079 V=10.0  +MOVJ EC00059 VJ=100.00
SFTOF
SFTON P043
MOVL C00080 BC00080 V=10.0  +MOVJ EC00060 VJ=100.00
MACRO1 MJ#(0) ARGF7
MOVL C00081 BC00081 V=10.0  +MOVJ EC00061 VJ=100.00
MOVL C00082 BC00082 V=10.0  +MOVJ EC00062 VJ=100.00
MOVL C00083 BC00083 V=10.0  +MOVJ EC00063 VJ=100.00
MOVL C00084 BC00084 V=10.0  +MOVJ EC00064 VJ=20.00
ARCOF
MOVJ C00085 BC00085 VJ=20.00  +MOVJ EC00065 VJ=20.00
SFTOF
MOVJ C00086 BC00086 VJ=100.00  +MOVJ EC00066 VJ=20.00
MOVJ C00087 BC00087 VJ=100.00  +MOVJ EC00067 VJ=20.00
SFTON P036
MOVJ C00088 BC00088 VJ=20.00  +MOVJ EC00068 VJ=100.00
ARCON
MOVL C00089 BC00089 V=10.0  +MOVJ EC00069 VJ=20.00
TIMER T=0.10
MOVL C00090 BC00090 V=8.3  +MOVJ EC00070 VJ=20.00
MOVL C00091 BC00091 V=8.3  +MOVJ EC00071 VJ=20.00
MOVL C00092 BC00092 V=10.0  +MOVJ EC00072 VJ=20.00
MOVL C00093 BC00093 V=10.0  +MOVJ EC00073 VJ=20.00
MOVL C00094 BC00094 V=10.0  +MOVJ EC00074 VJ=20.00
SFTOF
SFTON P040
MOVL C00095 BC00095 V=10.0  +MOVJ EC00075 VJ=20.00
MOVL C00096 BC00096 V=10.0  +MOVJ EC00076 VJ=20.00
SFTOF
SFTON P041
MOVL C00097 BC00097 V=10.0  +MOVJ EC00077 VJ=20.00
ARCON
MOVL C00098 BC00098 V=10.0  +MOVJ EC00078 VJ=20.00
MOVL C00099 BC00099 V=10.0  +MOVJ EC00079 VJ=50.00
MOVL C00100 BC00100 V=10.0  +MOVJ EC00080 VJ=15.00
ARCOF
MOVJ C00101 BC00101 VJ=15.00  +MOVJ EC00081 VJ=15.00
SFTOF
MOVJ C00102 BC00102 VJ=30.00  +MOVJ EC00082 VJ=30.00
SFTON P027
MOVJ C00103 BC00103 VJ=30.00  +MOVJ EC00083 VJ=30.00
ARCON
MOVL C00104 BC00104 V=10.0  +MOVJ EC00084 VJ=100.00
MOVL C00105 BC00105 V=10.0  +MOVJ EC00085 VJ=20.00
SFTOF
SFTON P026
MOVL C00106 BC00106 V=10.0  +MOVJ EC00086 VJ=20.00
MOVL C00107 BC00107 V=10.0  +MOVJ EC00087 VJ=20.00
ARCOF
SFTOF
MOVJ C00108 BC00108 VJ=100.00  +MOVJ EC00088 VJ=20.00
MOVJ C00109 BC00109 VJ=30.00  +MOVJ EC00089 VJ=30.00
MOVJ C00110 BC00110 VJ=100.00  +MOVJ EC00090 VJ=20.00
MOVJ C00111 BC00111 VJ=30.00  +MOVJ EC00091 VJ=30.00
SFTON P029
MOVJ C00112 BC00112 VJ=30.00  +MOVJ EC00092 VJ=30.00
ARCON
MOVL C00113 BC00113 V=10.0  +MOVJ EC00093 VJ=20.00
MOVL C00114 BC00114 V=10.0  +MOVJ EC00094 VJ=20.00
SFTOF
SFTON P030
MOVL C00115 BC00115 V=10.0  +MOVJ EC00095 VJ=20.00
MOVL C00116 BC00116 V=10.0  +MOVJ EC00096 VJ=20.00
MOVL C00117 BC00117 V=10.0  +MOVJ EC00097 VJ=20.00
ARCOF
MOVJ C00118 BC00118 VJ=20.00  +MOVJ EC00098 VJ=20.00
SFTOF
MOVJ C00119 BC00119 VJ=100.00  +MOVJ EC00099 VJ=100.00
MOVJ C00120 BC00120 VJ=100.00  +MOVJ EC00100 VJ=100.00
CALL JOB:CLEAN-R1_LONG
MOVJ C00121 BC00121 VJ=100.00  +MOVJ EC00101 VJ=100.00
MOVJ C00122 BC00122 VJ=100.00  +MOVJ EC00102 VJ=100.00
'SZUKANIE DRUGA STRONA
MOVJ C00123 BC00123 VJ=30.00  +MOVJ EC00103 VJ=15.00
SFTOF
MOVL C00124 BC00124 V=83.3  +MOVJ EC00104 VJ=15.00
REFP 3 RB1 C00125 BC00125
CALL JOB:SEARCH-R1
SET P035 P006
SFTON P035
MOVL C00126 BC00126 V=83.3  +MOVJ EC00105 VJ=15.00
REFP 3 RB1 C00127 BC00127
CALL JOB:SEARCH-R1
SET P035 P006
MOVL C00128 BC00128 V=83.3  +MOVJ EC00106 VJ=15.00
SFTOF
MOVJ C00129 BC00129 VJ=50.00  +MOVJ EC00107 VJ=50.00
MOVJ C00130 BC00130 VJ=15.00  +MOVJ EC00108 VJ=15.00
MOVL C00131 BC00131 V=83.3  +MOVJ EC00109 VJ=15.00
MOVL C00132 BC00132 V=83.3  +MOVJ EC00110 VJ=15.00
REFP 3 RB1 C00133 BC00133
CALL JOB:SEARCH-R1
SET P026 P006
SFTON P026
MOVL C00134 BC00134 V=83.3  +MOVJ EC00111 VJ=15.00
REFP 3 RB1 C00135 BC00135
CALL JOB:SEARCH-R1
SET P026 P006
MOVL C00136 BC00136 V=83.3  +MOVJ EC00112 VJ=15.00
SFTOF
MOVL C00137 BC00137 V=83.3  +MOVJ EC00113 VJ=15.00
MOVL C00138 BC00138 V=83.3  +MOVJ EC00114 VJ=15.00
REFP 3 RB1 C00139 BC00139
CALL JOB:SEARCH-R1
SET P027 P006
SFTON P027
MOVL C00140 BC00140 V=83.3  +MOVJ EC00115 VJ=15.00
REFP 3 RB1 C00141 BC00141
CALL JOB:SEARCH-R1
SET P027 P006
MOVL C00142 BC00142 V=83.3  +MOVJ EC00116 VJ=15.00
SFTOF
MOVL C00143 BC00143 V=83.3  +MOVJ EC00117 VJ=15.00
MOVL C00144 BC00144 V=83.3  +MOVJ EC00118 VJ=15.00
REFP 3 RB1 C00145 BC00145
CALL JOB:SEARCH-R1
SET P028 P006
SFTON P028
MOVL C00146 BC00146 V=83.3  +MOVJ EC00119 VJ=15.00
REFP 3 RB1 C00147 BC00147
CALL JOB:SEARCH-R1
SET P028 P006
MOVL C00148 BC00148 V=83.3  +MOVJ EC00120 VJ=15.00
SFTOF
MOVJ C00149 BC00149 VJ=15.00  +MOVJ EC00121 VJ=15.00
MOVJ C00150 BC00150 VJ=15.00  +MOVJ EC00122 VJ=15.00
SFTOF
MOVJ C00151 BC00151 VJ=15.00  +MOVJ EC00123 VJ=15.00
MOVL C00152 BC00152 V=83.3  +MOVJ EC00124 VJ=15.00
REFP 3 RB1 C00153 BC00153
CALL JOB:SEARCH-R1
SET P034 P006
SFTON P034
MOVL C00154 BC00154 V=83.3  +MOVJ EC00125 VJ=15.00
REFP 3 RB1 C00155 BC00155
CALL JOB:SEARCH-R1
SET P034 P006
MOVL C00156 BC00156 V=83.3  +MOVJ EC00126 VJ=15.00
MOVJ C00157 BC00157 VJ=15.00  +MOVJ EC00127 VJ=15.00
'KONIEC SZUKANIE DRUGA STRONA
'SPAWANIE DRUGA STRONA
MOVJ C00158 BC00158 VJ=15.00  +MOVJ EC00128 VJ=15.00
MACRO1 MJ#(0) ARGF7
SFTOF
SFTON P034
MOVJ C00159 BC00159 VJ=15.00  +MOVJ EC00129 VJ=15.00
ARCON
MOVL C00160 BC00160 V=10.0  +MOVJ EC00130 VJ=15.00
MOVL C00161 BC00161 V=10.0  +MOVJ EC00131 VJ=15.00
SFTOF
ARCOF
MOVJ C00162 BC00162 VJ=15.00  +MOVJ EC00132 VJ=15.00
MOVJ C00163 BC00163 VJ=50.00  +MOVJ EC00133 VJ=15.00
MOVJ C00164 BC00164 VJ=50.00  +MOVJ EC00134 VJ=50.00
MOVJ C00165 BC00165 VJ=50.00  +MOVJ EC00135 VJ=50.00
MOVJ C00166 BC00166 VJ=50.00  +MOVJ EC00136 VJ=50.00
SFTON P035
MOVL C00167 BC00167 V=83.3  +MOVJ EC00137 VJ=50.00
ARCON
MOVL C00168 BC00168 V=10.0  +MOVJ EC00138 VJ=50.00
MOVL C00169 BC00169 V=10.0  +MOVJ EC00139 VJ=50.00
ARCOF
SFTOF
MOVJ C00170 BC00170 VJ=20.00  +MOVJ EC00140 VJ=50.00
MOVJ C00171 BC00171 VJ=50.00  +MOVJ EC00141 VJ=20.00
SFTON P027
MOVJ C00172 BC00172 VJ=20.00  +MOVJ EC00142 VJ=20.00
ARCON
MOVL C00173 BC00173 V=9.2  +MOVJ EC00143 VJ=15.00
MOVL C00174 BC00174 V=9.2  +MOVJ EC00144 VJ=15.00
SFTOF
SFTON P028
MOVL C00175 BC00175 V=10.0  +MOVJ EC00145 VJ=15.00
ARCOF
MOVJ C00176 BC00176 VJ=20.00  +MOVJ EC00146 VJ=100.00
MOVJ C00177 BC00177 VJ=15.00  +MOVJ EC00147 VJ=15.00
SFTOF
MOVJ C00178 BC00178 VJ=15.00  +MOVJ EC00148 VJ=15.00
MOVJ C00179 BC00179 VJ=20.00  +MOVJ EC00149 VJ=20.00
SFTON P027
MOVJ C00180 BC00180 VJ=20.00  +MOVJ EC00150 VJ=20.00
ARCON
MOVL C00181 BC00181 V=10.0  +MOVJ EC00151 VJ=15.00
MOVL C00182 BC00182 V=10.0  +MOVJ EC00152 VJ=15.00
SFTOF
SFTON P026
MOVL C00183 BC00183 V=10.0  +MOVJ EC00153 VJ=15.00
MOVL C00184 BC00184 V=10.0  +MOVJ EC00154 VJ=15.00
ARCOF
MOVJ C00185 BC00185 VJ=15.00  +MOVJ EC00155 VJ=15.00
SFTOF
MOVJ C00186 BC00186 VJ=100.00  +MOVJ EC00156 VJ=15.00
MOVJ C00187 BC00187 VJ=100.00  +MOVJ EC00157 VJ=100.00
MOVJ C00188 BC00188 VJ=100.00  +MOVJ EC00158 VJ=100.00
MOVJ C00189 BC00189 VJ=100.00  +MOVJ EC00159 VJ=100.00
CALL JOB:CLEAN-R1_LONG
MOVJ C00190 BC00190 VJ=100.00  +MOVJ EC00160 VJ=100.00
MOVJ C00191 BC00191 VJ=100.00  +MOVJ EC00161 VJ=100.00
MOVJ C00192 BC00192 VJ=100.00  +MOVJ EC00162 VJ=100.00
MOVL C00193 BC00193 V=83.3  +MOVJ EC00163 VJ=15.00
REFP 3 RB1 C00194 BC00194
CALL JOB:SEARCH-R1
SET P021 P006
SFTON P021
MOVL C00195 BC00195 V=83.3  +MOVJ EC00164 VJ=15.00
REFP 3 RB1 C00196 BC00196
CALL JOB:SEARCH-R1
SET P021 P006
MOVL C00197 BC00197 V=83.3  +MOVJ EC00165 VJ=15.00
SFTOF
MOVL C00198 BC00198 V=166.7  +MOVJ EC00166 VJ=15.00
MOVL C00199 BC00199 V=83.3  +MOVJ EC00167 VJ=15.00
REFP 3 RB1 C00200 BC00200
CALL JOB:SEARCH-R1
SET P022 P006
SFTON P022
MOVL C00201 BC00201 V=83.3  +MOVJ EC00168 VJ=15.00
REFP 3 RB1 C00202 BC00202
CALL JOB:SEARCH-R1
SET P022 P006
MOVL C00203 BC00203 V=83.3  +MOVJ EC00169 VJ=15.00
SFTOF
MOVL C00204 BC00204 V=166.7  +MOVJ EC00170 VJ=15.00
MOVL C00205 BC00205 V=83.3  +MOVJ EC00171 VJ=15.00
REFP 3 RB1 C00206 BC00206
CALL JOB:SEARCH-R1
SET P023 P006
SFTON P023
MOVL C00207 BC00207 V=83.3  +MOVJ EC00172 VJ=15.00
REFP 3 RB1 C00208 BC00208
CALL JOB:SEARCH-R1
SET P023 P006
MOVL C00209 BC00209 V=83.3  +MOVJ EC00173 VJ=15.00
SFTOF
MOVL C00210 BC00210 V=166.7  +MOVJ EC00174 VJ=15.00
MOVL C00211 BC00211 V=83.3  +MOVJ EC00175 VJ=15.00
REFP 3 RB1 C00212 BC00212
CALL JOB:SEARCH-R1
SET P024 P006
SFTON P024
MOVL C00213 BC00213 V=83.3  +MOVJ EC00176 VJ=15.00
REFP 3 RB1 C00214 BC00214
CALL JOB:SEARCH-R1
SET P024 P006
MOVL C00215 BC00215 V=83.3  +MOVJ EC00177 VJ=15.00
SFTOF
MOVL C00216 BC00216 V=166.7  +MOVJ EC00178 VJ=15.00
MOVL C00217 BC00217 V=83.3  +MOVJ EC00179 VJ=15.00
REFP 3 RB1 C00218 BC00218
CALL JOB:SEARCH-R1
SET P025 P006
SFTON P025
MOVL C00219 BC00219 V=83.3  +MOVJ EC00180 VJ=15.00
REFP 3 RB1 C00220 BC00220
CALL JOB:SEARCH-R1
SET P025 P006
MOVL C00221 BC00221 V=133.3  +MOVJ EC00181 VJ=15.00
SFTOF
MOVJ C00222 BC00222 VJ=30.00  +MOVJ EC00182 VJ=100.00
MOVJ C00223 BC00223 VJ=30.00  +MOVJ EC00183 VJ=30.00
SFTON P023
MACRO1 MJ#(0) ARGF7
MOVL C00224 BC00224 V=83.3  +MOVJ EC00184 VJ=30.00
ARCON
SFTOF
SFTON P022
MOVL C00225 BC00225 V=10.8  +MOVJ EC00185 VJ=30.00
SFTOF
SFTON P021
MOVL C00226 BC00226 V=10.8  +MOVJ EC00186 VJ=30.00
MOVL C00227 BC00227 V=10.8  +MOVJ EC00187 VJ=30.00
ARCOF
SFTOF
MOVJ C00228 BC00228 VJ=30.00  +MOVJ EC00188 VJ=30.00
MOVJ C00229 BC00229 VJ=30.00  +MOVJ EC00189 VJ=30.00
SFTON P023
MOVL C00230 BC00230 V=83.3  +MOVJ EC00190 VJ=30.00
ARCON
SFTOF
SFTON P024
MOVL C00231 BC00231 V=10.8  +MOVJ EC00191 VJ=30.00
SFTOF
SFTON P025
MOVL C00232 BC00232 V=10.8  +MOVJ EC00192 VJ=30.00
MOVL C00233 BC00233 V=10.8  +MOVJ EC00193 VJ=30.00
MOVL C00234 BC00234 V=10.8  +MOVJ EC00194 VJ=30.00
ARCOF
SFTOF
MOVJ C00235 BC00235 VJ=30.00  +MOVJ EC00195 VJ=30.00
MOVJ C00236 BC00236 VJ=30.00  +MOVJ EC00196 VJ=30.00
MOVJ C00237 BC00237 VJ=100.00  +MOVJ EC00197 VJ=100.00
MOVJ C00238 BC00238 VJ=30.00  +MOVJ EC00198 VJ=30.00
CALL JOB:ONLYCUT-R1_LONG
MOVJ C00239 BC00239 VJ=30.00  +MOVJ EC00199 VJ=30.00
MOVJ C00240 BC00240 VJ=100.00  +MOVJ EC00200 VJ=100.00
MOVJ C00241 BC00241 VJ=60.00  +MOVJ EC00201 VJ=30.00
MOVJ C00242 BC00242 VJ=60.00  +MOVJ EC00202 VJ=30.00
MOVJ C00243 BC00243 VJ=60.00  +MOVJ EC00203 VJ=30.00
MOVJ C00244 BC00244 VJ=60.00  +MOVJ EC00204 VJ=30.00
MOVJ C00245 BC00245 VJ=100.00  +MOVJ EC00205 VJ=100.00
MOVL C00246 BC00246 V=83.3  +MOVJ EC00206 VJ=15.00
REFP 3 RB1 C00247 BC00247
CALL JOB:SEARCH-R1
SET P021 P006
SFTON P021
MOVL C00248 BC00248 V=83.3  +MOVJ EC00207 VJ=15.00
REFP 3 RB1 C00249 BC00249
CALL JOB:SEARCH-R1
SET P021 P006
MOVL C00250 BC00250 V=83.3  +MOVJ EC00208 VJ=15.00
SFTOF
MOVL C00251 BC00251 V=166.7  +MOVJ EC00209 VJ=15.00
MOVL C00252 BC00252 V=83.3  +MOVJ EC00210 VJ=15.00
REFP 3 RB1 C00253 BC00253
CALL JOB:SEARCH-R1
SET P022 P006
SFTON P022
MOVL C00254 BC00254 V=83.3  +MOVJ EC00211 VJ=15.00
REFP 3 RB1 C00255 BC00255
CALL JOB:SEARCH-R1
SET P022 P006
MOVL C00256 BC00256 V=83.3  +MOVJ EC00212 VJ=15.00
SFTOF
MOVL C00257 BC00257 V=166.7  +MOVJ EC00213 VJ=15.00
MOVL C00258 BC00258 V=83.3  +MOVJ EC00214 VJ=15.00
REFP 3 RB1 C00259 BC00259
CALL JOB:SEARCH-R1
SET P023 P006
SFTON P023
MOVL C00260 BC00260 V=83.3  +MOVJ EC00215 VJ=15.00
REFP 3 RB1 C00261 BC00261
CALL JOB:SEARCH-R1
SET P023 P006
MOVL C00262 BC00262 V=83.3  +MOVJ EC00216 VJ=15.00
SFTOF
MOVL C00263 BC00263 V=166.7  +MOVJ EC00217 VJ=15.00
MOVL C00264 BC00264 V=83.3  +MOVJ EC00218 VJ=15.00
REFP 3 RB1 C00265 BC00265
CALL JOB:SEARCH-R1
SET P024 P006
SFTON P024
MOVL C00266 BC00266 V=83.3  +MOVJ EC00219 VJ=15.00
REFP 3 RB1 C00267 BC00267
CALL JOB:SEARCH-R1
SET P024 P006
MOVL C00268 BC00268 V=83.3  +MOVJ EC00220 VJ=15.00
SFTOF
MOVL C00269 BC00269 V=166.7  +MOVJ EC00221 VJ=15.00
MOVL C00270 BC00270 V=83.3  +MOVJ EC00222 VJ=15.00
REFP 3 RB1 C00271 BC00271
CALL JOB:SEARCH-R1
SET P025 P006
SFTON P025
MOVL C00272 BC00272 V=83.3  +MOVJ EC00223 VJ=15.00
REFP 3 RB1 C00273 BC00273
CALL JOB:SEARCH-R1
SET P025 P006
MOVL C00274 BC00274 V=83.3  +MOVJ EC00224 VJ=15.00
SFTOF
MOVJ C00275 BC00275 VJ=30.00  +MOVJ EC00225 VJ=100.00
MOVJ C00276 BC00276 VJ=30.00  +MOVJ EC00226 VJ=30.00
SFTON P023
MOVL C00277 BC00277 V=83.3  +MOVJ EC00227 VJ=30.00
ARCON
SFTOF
SFTON P022
MOVL C00278 BC00278 V=10.8  +MOVJ EC00228 VJ=30.00
SFTOF
SFTON P021
MOVL C00279 BC00279 V=10.8  +MOVJ EC00229 VJ=30.00
MOVL C00280 BC00280 V=10.8  +MOVJ EC00230 VJ=30.00
ARCOF
SFTOF
MOVJ C00281 BC00281 VJ=30.00  +MOVJ EC00231 VJ=30.00
MOVJ C00282 BC00282 VJ=30.00  +MOVJ EC00232 VJ=30.00
SFTON P023
MOVL C00283 BC00283 V=83.3  +MOVJ EC00233 VJ=30.00
ARCON
SFTOF
SFTON P024
MOVL C00284 BC00284 V=10.8  +MOVJ EC00234 VJ=30.00
SFTOF
SFTON P025
MOVL C00285 BC00285 V=10.8  +MOVJ EC00235 VJ=30.00
MOVL C00286 BC00286 V=10.8  +MOVJ EC00236 VJ=30.00
MOVL C00287 BC00287 V=10.8  +MOVJ EC00237 VJ=30.00
ARCOF
SFTOF
MOVJ C00288 BC00288 VJ=50.00  +MOVJ EC00238 VJ=30.00
MOVJ C00289 BC00289 VJ=50.00  +MOVJ EC00239 VJ=30.00
MOVJ C00290 BC00290 VJ=50.00  +MOVJ EC00240 VJ=30.00
MOVJ C00291 BC00291 VJ=100.00  +MOVJ EC00241 VJ=100.00
DOUT OT#(1433) OFF
DOUT OT#(1435) OFF
PAUSE
PAUSE
'ZALOZYC USZY ZE SCIANY
MOVJ C00292 BC00292 VJ=100.00  +MOVJ EC00242 VJ=100.00
END
